// TIA Portal V20 export
FUNCTION_BLOCK "FB_Tracability"   // FB700, SCL
{ S7_Optimized_Access := 'TRUE' }
// stored: AutoNumber false, MemoryReserve 100, SetENOAutomatically false
   VAR_INPUT
      iCondTransfertExtInTo1 : Bool;
      iCondTransfertExtInTo2 : Bool;
      iCondTransfert1To3 : Bool;
      iCondTransfert2To3 : Bool;
      iCondTransfert3To4 : Bool;
      iCondTransfert4To5 : Bool;
      iCondTransfert5To6 : Bool;
      iCondTransfert5To7 : Bool;
      iCondTransfert6ToExtOut : Bool;
      iCondTransfert7ToExtOut : Bool;
   END_VAR
   VAR
      sRT_ConditionExtInTo1 : R_TRIG;
      sRT_ConditionExtInTo2 { S7_SetPoint := 'True'} : R_TRIG;
      sRT_Condition1To3 { S7_SetPoint := 'True'} : R_TRIG;
      sRT_Condition2To3 { S7_SetPoint := 'True'} : R_TRIG;
      sRT_Condition3To4 { S7_SetPoint := 'True'} : R_TRIG;
      sRT_Condition4To5 { S7_SetPoint := 'True'} : R_TRIG;
      sRT_Condition5To6 { S7_SetPoint := 'True'} : R_TRIG;
      sRT_Condition5To7 { S7_SetPoint := 'True'} : R_TRIG;
      sRT_Condition6ToExtOut { S7_SetPoint := 'True'} : R_TRIG;
      sRT_Condition7ToExtOut { S7_SetPoint := 'True'} : R_TRIG;
      sIndex : Int;
      sCheckTransfertExtInTo1 : Bool;
      sCheckTransfertExtInTo2 : Bool;
      sCheckTransfert1To3 : Bool;
      sCheckTransfert2To3 : Bool;
      sCheckTransfert3To4 : Bool;
      sCheckTransfert4To5 : Bool;
      sCheckTransfert5To6 : Bool;
      sCheckTransfert5To7 : Bool;
      sCheckTransfert6ToExtOut : Bool;
      sCheckTransfert7ToExtOut : Bool;
      sLaserTime : "FB_TimeCounter";
      sMemoPartDMC { S7_SetPoint := 'True'} : Array[0..19] of Byte;
   END_VAR
   VAR RETAIN
      sIEC_CounterCycleLaser { S7_SetPoint := 'True'} : TONR_TIME;
      sIEC_CounterCycleTime { S7_SetPoint := 'True'} : TONR_TIME;
      sStartCounterCycleLaser { S7_SetPoint := 'True'} : Bool;
      sStartCounterCycleTime { S7_SetPoint := 'True'} : Bool;
   END_VAR
   VAR_TEMP
      tFailCodePart : Int;
      tFailCodeBackwall : Int;
      tHoleNumber : Int;
      tMeasureZ : Real;
      tWOZ : Int;
      tWOC : Int;
      tTotalCycleTimeCh1 : Int;
      tLaserCycleTimeCh1 : Int;
   END_VAR
   VAR CONSTANT
      POSITION_NUMBER : Int := 7;
   END_VAR
BEGIN
   REGION Reset data Postions station 1
       // Positions :
           //  1 : Shuttle 1 Undrilled Part
           //  2 : Shuttle 2 Undrilled Part
           //  3 : Gripper   Undrilled Part
           //  4 : Fixture
           //  5 : Gripper   Drilled Part
           //  6 : Shuttle 1 Drilled Part
           //  7 : Shuttle 2 Drilled Part

       IF "LBP_Chan1".A_Ref THEN
           #sCheckTransfertExtInTo1 := FALSE;     
           #sCheckTransfertExtInTo2 := FALSE;     
           #sCheckTransfert1To3 := FALSE;            
           #sCheckTransfert2To3 := FALSE;           
           #sCheckTransfert3To4 := FALSE;           
           #sCheckTransfert4To5 := FALSE;            
           #sCheckTransfert5To6 := FALSE;        
           #sCheckTransfert5To7 := FALSE;         
           #sCheckTransfert6ToExtOut := FALSE;   
           #sCheckTransfert7ToExtOut := FALSE;     
           FOR #sIndex := 0 TO #POSITION_NUMBER DO
               "FC_ResetPositionData"(iDataPosition := #sIndex);
           END_FOR;
       END_IF;
   END_REGION

   REGION Transfert Postions data station 1 
       IF #sCheckTransfert1To3 THEN
           // Transfert data from position 1 To 3 - Shuttle 1 to Loading Gripper 
           "DB_DataPositions".Position[3] := "DB_DataPositions".Position[1];
           // Reset data in position 1
           "FC_ResetPositionData"(iDataPosition := 1);
           #sCheckTransfert1To3 := FALSE;
       END_IF;

       IF #sCheckTransfert2To3 THEN
           // Transfert data from position 2 To 3 - Shuttle 2 to Loading Gripper 
           "DB_DataPositions".Position[3] := "DB_DataPositions".Position[2];
           // Reset data in position 2
           "FC_ResetPositionData"(iDataPosition := 2);
           #sCheckTransfert2To3 := FALSE;
       END_IF;

       IF #sCheckTransfert3To4 THEN
           // Transfert data from position 3 To 4 - Loading Gripper to Fixture
           "DB_DataPositions".Position[4] := "DB_DataPositions".Position[3];
           // Reset data in position 3
           "FC_ResetPositionData"(iDataPosition := 3);
           #sCheckTransfert3To4 := FALSE;
       END_IF;

       IF #sCheckTransfert4To5 THEN
           // Transfert data from position 4 To 5 - Fixture to Unloading Gripper
           "DB_DataPositions".Position[5] := "DB_DataPositions".Position[4];
           // Reset data in position 4
           "FC_ResetPositionData"(iDataPosition := 4);
           #sCheckTransfert4To5 := FALSE;
       END_IF;

       IF #sCheckTransfert5To6 THEN
           // Transfert data from position 5 To 6 - Unloading Gripper to Shuttle 1
           "DB_DataPositions".Position[6] := "DB_DataPositions".Position[5];
           // Reset data in position 5
           "FC_ResetPositionData"(iDataPosition := 5);
           #sCheckTransfert5To6 := FALSE;
       END_IF;

       IF #sCheckTransfert5To7 THEN
           // Transfert data from position 5 To 7 - Unloading Gripper to Shuttle 2
           "DB_DataPositions".Position[7] := "DB_DataPositions".Position[5];
           // Reset data in position 5
           "FC_ResetPositionData"(iDataPosition := 5);
           #sCheckTransfert5To7 := FALSE;
       END_IF;

       IF #sCheckTransfert6ToExtOut THEN
           // Shift of the the array for the new final part
           FOR #sIndex := 98 TO 0 BY -1 DO
               "DB_DataFinalPart".FinalPart[#sIndex + 1] := "DB_DataFinalPart".FinalPart[#sIndex];
           END_FOR;
           // Transfert data from position 6 TO the DB final part - Shuttle 1 to DB final part
           "DB_DataFinalPart".FinalPart[0] := "DB_DataPositions".Position[6];
           "FC_ResetPositionData"(iDataPosition := 6);
           #sCheckTransfert6ToExtOut := FALSE;
       END_IF;

       IF #sCheckTransfert7ToExtOut THEN
           // Shift of the the array for the new final part
           FOR #sIndex := 98 TO 0 BY -1 DO
               "DB_DataFinalPart".FinalPart[#sIndex + 1] := "DB_DataFinalPart".FinalPart[#sIndex];
           END_FOR;
           // Transfert data from position 7 TO the DB final part - Shuttle 2 to DB final part
           "DB_DataFinalPart".FinalPart[0] := "DB_DataPositions".Position[7];
           "FC_ResetPositionData"(iDataPosition := 7);
           #sCheckTransfert7ToExtOut := FALSE;
       END_IF;
   END_REGION

   REGION Condition for the Transfert Postions data
       // Conditions from Ext To position 1 - External Loader to Shuttle 1
       #sRT_ConditionExtInTo1(CLK := #iCondTransfertExtInTo1);
       IF #sRT_ConditionExtInTo1.Q THEN
           #sCheckTransfertExtInTo1 := TRUE;
       END_IF;

       // Conditions from Ext To position 2 - External Loader to Shuttle 2
       #sRT_ConditionExtInTo2(CLK := #iCondTransfertExtInTo2);
       IF #sRT_ConditionExtInTo2.Q THEN
           #sCheckTransfertExtInTo2 := TRUE;
       END_IF;

       // Conditions from position 1 To 3 - Shuttle 1 to Loading Gripper 
       #sRT_Condition1To3(CLK:=#iCondTransfert1To3);
       IF #sRT_Condition1To3.Q THEN
           #sCheckTransfert1To3 := TRUE;
       END_IF;

       // Conditions from position 2 To 3 - Shuttle 2 to Loading Gripper 
       #sRT_Condition2To3(CLK := #iCondTransfert2To3);
       IF #sRT_Condition2To3.Q THEN
           #sCheckTransfert2To3 := TRUE;
       END_IF;

       // Conditions from position 3 To 4 - Loading Gripper to Fixture
       #sRT_Condition3To4(CLK := #iCondTransfert3To4);
       IF #sRT_Condition3To4.Q THEN
           #sCheckTransfert3To4 := TRUE;
       END_IF;

       // Conditions from position 4 To 5 - Fixture to Unloading Gripper
       #sRT_Condition4To5(CLK := #iCondTransfert4To5);
       IF #sRT_Condition4To5.Q THEN
           #sCheckTransfert4To5 := TRUE;
       END_IF;

       // Conditions from position 5 To 6 - Unloading Gripper to Shuttle 1
       #sRT_Condition5To6(CLK := #iCondTransfert5To6);
       IF #sRT_Condition5To6.Q THEN
           #sCheckTransfert5To6 := TRUE;
       END_IF;

       // Conditions from position 5 To 7 - Unloading Gripper to Shuttle 2
       #sRT_Condition5To7(CLK := #iCondTransfert5To7);
       IF #sRT_Condition5To7.Q THEN
           #sCheckTransfert5To7 := TRUE;
       END_IF;

       // Conditions from position 6 To Ext - Shuttle 1 to External Loader
       #sRT_Condition6ToExtOut(CLK := #iCondTransfert6ToExtOut);
       IF #sRT_Condition6ToExtOut.Q THEN
           #sCheckTransfert6ToExtOut := TRUE;
       END_IF;

       // Conditions from position 7 To Ext - Shuttle 2 to External Loader
       #sRT_Condition7ToExtOut(CLK := #iCondTransfert7ToExtOut);
       IF #sRT_Condition7ToExtOut.Q THEN
           #sCheckTransfert7ToExtOut := TRUE;
       END_IF;
   END_REGION

   REGION Update Data
       // Détection nouvelle pièce
       IF #sCheckTransfertExtInTo1 THEN
           // Initialisation de la donnée de la pièce sur shuttle 1
           "DB_DataPositions".Position[1].DMC := "DB_SonplasMain".sSonplasLoader.iPartInDMC_CodeShuttle1;
           #sCheckTransfertExtInTo1 := FALSE;
       END_IF;
       IF #sCheckTransfertExtInTo2 THEN
           // Initialisation de la donnée de la pièce sur shuttle 2
           "DB_DataPositions".Position[2].DMC := "DB_SonplasMain".sSonplasLoader.iPartInDMC_CodeShuttle2;
           #sCheckTransfertExtInTo2 := FALSE;
       END_IF;
       // Fail code part
       IF "LBP_Chan1".MDyn[69] THEN
           #tFailCodePart := REAL_TO_INT("LBP_Chan1".H1);
       END_IF;
       // Measure Z
       IF "LBP_Chan1".MDyn[98] THEN
           #tHoleNumber := REAL_TO_INT("LBP_Chan1".H1);
           #tMeasureZ := "LBP_Chan1".H2;
       END_IF;
       // WOZ
       IF "LBP_Chan1".MDyn[37] THEN
           #tWOZ := REAL_TO_INT("LBP_Chan1".H1);
       END_IF;
       // WOC
       IF "LBP_Chan1".MDyn[38] THEN
           #tWOC := REAL_TO_INT("LBP_Chan1".H1);
       END_IF;
       "DB_DataPositions".Position[4].FailCode := #tFailCodePart;
       "DB_DataPositions".Position[4].WOZ_Measure := #tWOZ;
       "DB_DataPositions".Position[4].WOC_Measure := #tWOC;
       #sMemoPartDMC:= "DB_DataPositions".Position[4].DMC;
       // Counter if cycle time
       IF "LBP_Chan1".MDyn[72] THEN             // M72 : Start counter of cycle time
           #sStartCounterCycleTime := TRUE;
       ELSIF "LBP_Chan1".MDyn[73] THEN          // M73 : Stop counter of cycle time
           #sStartCounterCycleTime := FALSE;
       END_IF;
       #sIEC_CounterCycleTime(IN:=#sStartCounterCycleTime,
                              R:=NOT #sStartCounterCycleTime,
                              PT:=t#10m);
       // Counter of cycle laser
       IF "LBP_Chan1".MDyn[71] THEN            // M71 : Start calculation laser time 
           #sStartCounterCycleLaser := TRUE;
       ELSIF "LBP_Chan1".MDyn[68] THEN         // M68 : Set Lasered (Tracability)
           #sStartCounterCycleLaser := FALSE;
       END_IF;
       #sIEC_CounterCycleLaser(IN:=#sStartCounterCycleLaser,
                               R:=NOT #sStartCounterCycleLaser,
                               PT:=t#10m);
       // Mesure ZED Backwall PAS UTILISE SUR FL0153 A SUPPRIMER
       IF "LBP_Chan1".MDyn[29] THEN
           #tFailCodeBackwall := REAL_TO_INT("LBP_Chan1".H1);
       END_IF;
       // Close unload gripper
       IF "DB_DataPositions".Position[4].DMC = #sMemoPartDMC THEN
           IF "LBP_Chan1".MDyn[82] THEN
               "DB_DataPositions".Position[4].TotalCycleTime := TIME_TO_INT(#sIEC_CounterCycleTime.ET);
               "DB_DataPositions".Position[4].LaserCycleTime := TIME_TO_INT(#sIEC_CounterCycleLaser.ET);
           END_IF;
           "DB_DataPositions".Position[4].FailCodeBackwall := #tFailCodeBackwall;

       ELSIF "DB_DataPositions".Position[5].DMC = #sMemoPartDMC THEN
           IF "LBP_Chan1".MDyn[82] THEN
               "DB_DataPositions".Position[5].TotalCycleTime := TIME_TO_INT(#sIEC_CounterCycleTime.ET);
               "DB_DataPositions".Position[5].LaserCycleTime := TIME_TO_INT(#sIEC_CounterCycleLaser.ET);
           END_IF;
           "DB_DataPositions".Position[5].FailCodeBackwall := #tFailCodeBackwall;
       END_IF;
   END_REGION
END_FUNCTION_BLOCK
